FUNCTION NextStep : UDINT
VAR_INPUT
	StateVar	: UDINT;
END_VAR
VAR
END_VAR

NextStep := ((StateVar / 10)* 10) + 10;

END_FUNCTION

(* stored: Version 1.1.0.1, ProductVersion 3.1.4024.12
   POU NextStep: Id {4ab0e0b1-cc54-4466-88b3-4c3f17eb8b0c}, SpecialFunc None *)
